FUNCTION_BLOCK PICKER_HMI_NEW (* Composite Function Block Type *)
  (* Standard: 61499-2 *)
  (* Version 0.2, 2003-12-05, JHC, Rockwell Automation, Renamed from NEWCOMPFB. *)
  (* Version 0.1, 2002-01-08, JHC, Rockwell Automation, Added DLY FB as example. *)
  (* Version 0.0, 2000-05-27, JHC, Rockwell Automation *)
  (* Compiler header: package fb.rt.pnp;import fb.rt.hmi.*; *)
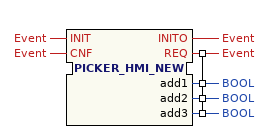
  EVENT_INPUT
    INIT;
    CNF; (* Confirmation from Plug *)
  END_EVENT
  EVENT_OUTPUT
    INITO;
    REQ WITH add1, add2, add3; (* Request from Socket *)
  END_EVENT
  VAR_OUTPUT
    add1 : BOOL;
    add2 : BOOL;
    add3 : BOOL;
  END_VAR
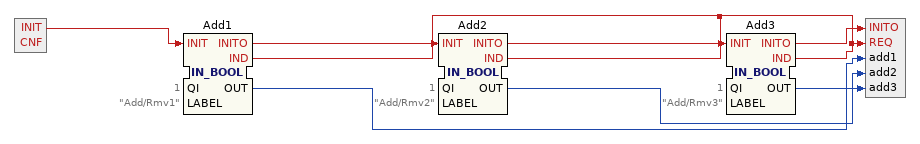
  FBS
    Add1 : IN_BOOL(QI := 1, LABEL := "Add/Rmv1");
    Add2 : IN_BOOL(QI := 1, LABEL := "Add/Rmv2");
    Add3 : IN_BOOL(QI := 1, LABEL := "Add/Rmv3");
  END_FBS
  EVENT_CONNECTIONS
    Add1.INITO TO Add2.INIT;
    Add2.INITO TO Add3.INIT;
    Add3.INITO TO INITO;
    Add1.IND TO REQ;
    Add2.IND TO REQ;
    Add3.IND TO REQ;
    INIT TO Add1.INIT;
  END_CONNECTIONS
  DATA_CONNECTIONS
    Add1.OUT TO add1;
    Add2.OUT TO add2;
    Add3.OUT TO add3;
  END_CONNECTIONS
END_FUNCTION_BLOCK
